// TIA Portal V17 export
// export: Created 2025-06-26T06:49:20.3674606Z, ExportSetting WithDefaults, DisplayName Totally Integrated Automation Portal, DisplayVersion V17 Update 8, DisplayName TIA Portal Openness, DisplayVersion V17 Update 8, DisplayName TIA Portal Version Control Interface, DisplayVersion V17, DisplayName STEP 7 Professional, DisplayVersion V17 Update 8, DisplayName STEP 7 Safety, DisplayVersion V17 Update 6, DisplayName WinCC Advanced, DisplayVersion V17 Update 8
DATA_BLOCK "S7_Internal_DB"   // DB1
VERSION : 0.1
// stored: AutoNumber false, DBAccessibleFromOPCUA true, InstanceOfName S7_Internal, InstanceOfType FB
"S7_Internal"
   // VAR_INPUT
   //    bEnable : Bool := true;
   // END_VAR
   // VAR
   //    nGroup : USInt;
   //    xGroup1 : Byte;
   //    xGroup2 : Byte;
   //    xGroup3 : Byte;
   //    xGroup4 : Byte;
   //    GET_1 { S7_SetPoint := 'True'} : GET;
   //    GET_2 { S7_SetPoint := 'True'} : GET;
   //    GET_3 { S7_SetPoint := 'True'} : GET;
   //    GET_AI_4 { S7_SetPoint := 'True'} : GET;
   //    GET_AI_5 { S7_SetPoint := 'True'} : GET;
   //    GET_AI_6 { S7_SetPoint := 'True'} : GET;
   //    GET_AI_7 { S7_SetPoint := 'True'} : GET;
   //    GET_AI_8 { S7_SetPoint := 'True'} : GET;
   //    PUT_1 { S7_SetPoint := 'True'} : PUT;
   //    CommCycles { S7_SetPoint := 'True'} : UDInt;
   //    Group1Timeout : TON_TIME;
   //    Group2Timeout { S7_SetPoint := 'True'} : TON_TIME;
   //    Group3Timeout { S7_SetPoint := 'True'} : TON_TIME;
   //    Group4Timeout { S7_SetPoint := 'True'} : TON_TIME;
   //    RuntimeMemory { S7_SetPoint := 'True'} : LReal;
   //    RuntimeElapsed : LReal;
   // END_VAR
BEGIN
END_DATA_BLOCK
